Staubli VAL3: MOTION.dtx

mdesc mNomSpeed
mdesc mRun
public num nAction[12 2]
public num nStartTraj
public num nEndTraj
public num nMoveidAction[12 2]
public string sMotionMess
bool bSync
num nTestBuff
bool bWeldAction
